FUNCTION_BLOCK FortePVForecaster (* Forte variant of the PVForecaste FB. *)
  (* Standard: 61499-2; Description: This function block creates a back up of its forecast data which can be re-loaded if the device has to restart. Otherwise, it is exactly the same as the PVForecaster FB. *)
  (* Version 1.0, 2017-09-10, Marc Jakobi, HTW Berlin *)
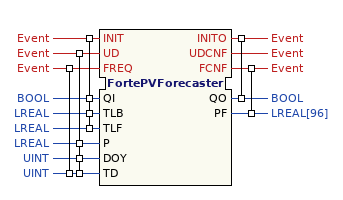
  EVENT_INPUT
    INIT WITH QI, TLB, TLF; (* Service Initialization *)
    UD WITH P, DOY, TD; (* PV Forecast Update Request *)
    FREQ WITH TD; (* Forecast Request *)
  END_EVENT
  EVENT_OUTPUT
    INITO WITH QO; (* Initialization Confirm *)
    UDCNF; (* Update Algorithm Execution Confirmation *)
    FCNF WITH PF; (* Forecast Confirmation *)
  END_EVENT
  VAR_INPUT
    QI : BOOL; (* Event Input Qualifier *)
    TLB : LREAL; (* Time frame to look back when generating forecasts in h *)
    TLF : LREAL; (* Time frame to forecast ahead (look forward) in h *)
    P : LREAL; (* Measured PV power in W *)
    DOY : UINT; (* Day of the year [1..365] *)
    TD : UINT; (* Time of day [min] [0..1439] *)
  END_VAR
  VAR_OUTPUT
    QO : BOOL; (* Event Output Qualifier *)
    PF : ARRAY [0..95] OF LREAL; (* Forecasted PV power *)
  END_VAR
  (* Service APPLICATION/RESOURCE: Forte variant of the PVForecaste FB. *)
END_FUNCTION_BLOCK
